# EPICS substitutions: adsApp/Db/adsGeneral.substitutions
file "adsGeneral.template"
{
pattern
{P,      PORT}
{ADSTEST:,  ADS_1}
}
